// TIA Portal V20 export
FUNCTION "左顶升伺服" : Void   // FC1, LAD
{ S7_Optimized_Access := 'TRUE' }
// stored: SetENOAutomatically false
BEGIN

REGION Network 1 (SCL)
   "左顶升IS620F控制字".%X0 := "1200_下载".位1;
   "左顶升IS620F控制字".%X1 := "1200_下载".位2;
   "左顶升IS620F控制字".%X2 := "1200_下载".位3;
   "左顶升IS620F控制字".%X3 := "1200_下载".位4;
   "左顶升IS620F控制字".%X4 := "1200_下载".位5;
   "左顶升IS620F控制字".%X5 := "1200_下载".位6;
   "左顶升IS620F控制字".%X6 := "1200_下载".位7;
   "左顶升IS620F控制字".%X7 := "1200_下载".位8;

   "左_回原模式" := "1200_下载".整型1;

   "左_绝对位置" := "1200_下载".浮点数1;
   "左_绝对速度" := "1200_下载".浮点数2;
   "左_相对位置" := "1200_下载".浮点数3;
   "左_相对速度" := "1200_下载".浮点数4;
   "左_点动速度" := "1200_下载".浮点数5;
END_REGION

REGION Network 2
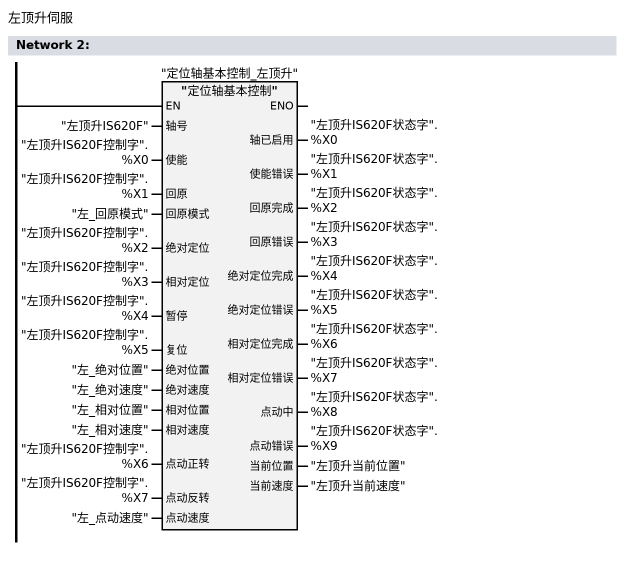
   RUNG wire#powerrail
      "定位轴基本控制_左顶升"(轴号 := "左顶升IS620F", 使能 := "左顶升IS620F控制字".%X0, 回原 := "左顶升IS620F控制字".%X1, 回原模式 := "左_回原模式", 绝对定位 := "左顶升IS620F控制字".%X2, 相对定位 := "左顶升IS620F控制字".%X3, 暂停 := "左顶升IS620F控制字".%X4, 复位 := "左顶升IS620F控制字".%X5, 绝对位置 := "左_绝对位置", 绝对速度 := "左_绝对速度", 相对位置 := "左_相对位置", 相对速度 := "左_相对速度", 点动正转 := "左顶升IS620F控制字".%X6, 点动反转 := "左顶升IS620F控制字".%X7, 点动速度 := "左_点动速度", 轴已启用 => "左顶升IS620F状态字".%X0, 使能错误 => "左顶升IS620F状态字".%X1, 回原完成 => "左顶升IS620F状态字".%X2, 回原错误 => "左顶升IS620F状态字".%X3, 绝对定位完成 => "左顶升IS620F状态字".%X4, 绝对定位错误 => "左顶升IS620F状态字".%X5, 相对定位完成 => "左顶升IS620F状态字".%X6, 相对定位错误 => "左顶升IS620F状态字".%X7, 点动中 => "左顶升IS620F状态字".%X8, 点动错误 => "左顶升IS620F状态字".%X9, 当前位置 => "左顶升当前位置", 当前速度 => "左顶升当前速度")
   END_RUNG
   // the same network as SCL:
   "定位轴基本控制_左顶升"(轴号 := "左顶升IS620F",   // "定位轴基本控制"
                 使能 := "左顶升IS620F控制字".%X0,
                 回原 := "左顶升IS620F控制字".%X1,
                 回原模式 := "左_回原模式",
                 绝对定位 := "左顶升IS620F控制字".%X2,
                 相对定位 := "左顶升IS620F控制字".%X3,
                 暂停 := "左顶升IS620F控制字".%X4,
                 复位 := "左顶升IS620F控制字".%X5,
                 绝对位置 := "左_绝对位置",
                 绝对速度 := "左_绝对速度",
                 相对位置 := "左_相对位置",
                 相对速度 := "左_相对速度",
                 点动正转 := "左顶升IS620F控制字".%X6,
                 点动反转 := "左顶升IS620F控制字".%X7,
                 点动速度 := "左_点动速度",
                 轴已启用 => "左顶升IS620F状态字".%X0,
                 使能错误 => "左顶升IS620F状态字".%X1,
                 回原完成 => "左顶升IS620F状态字".%X2,
                 回原错误 => "左顶升IS620F状态字".%X3,
                 绝对定位完成 => "左顶升IS620F状态字".%X4,
                 绝对定位错误 => "左顶升IS620F状态字".%X5,
                 相对定位完成 => "左顶升IS620F状态字".%X6,
                 相对定位错误 => "左顶升IS620F状态字".%X7,
                 点动中 => "左顶升IS620F状态字".%X8,
                 点动错误 => "左顶升IS620F状态字".%X9,
                 当前位置 => "左顶升当前位置",
                 当前速度 => "左顶升当前速度");
END_REGION

REGION Network 3 (SCL)
   "1200_上传".位1 := "左顶升IS620F状态字".%X0;
   "1200_上传".位2 := "左顶升IS620F状态字".%X1;
   "1200_上传".位3 := "左顶升IS620F状态字".%X2;
   "1200_上传".位4 := "左顶升IS620F状态字".%X3;
   "1200_上传".位5 := "左顶升IS620F状态字".%X4;
   "1200_上传".位6 := "左顶升IS620F状态字".%X5;
   "1200_上传".位7 := "左顶升IS620F状态字".%X6;
   "1200_上传".位8 := "左顶升IS620F状态字".%X7;
   "1200_上传".位9 := "左顶升IS620F状态字".%X8;
   "1200_上传".位10 := "左顶升IS620F状态字".%X9;

   "1200_上传".浮点数1 := "左顶升当前位置";
   "1200_上传".浮点数2 := "左顶升当前速度";
END_REGION
END_FUNCTION
